Staubli VAL3: FloatToBytes.pgx

program FloatToBytes(num valIn, num& hByte, num& lByte)
  local num int
begin
//*******************************************************************************
//*   ______
//*  / _____) /|
//* | |      / /
//* | | /\  / /
//* | | \ \/ /  _      Copyright (c) KEOLABS, 2016
//* | |  \__/  | |        http://www.keolabs.com
//* | |________| |
//*  \__________/
//*
//********************************************************************************
//*@file          : FloatToBytes
//*@author        : Yves Ragot
//*@version       : $Id: FloatToBytes.pgx 1558 2017-01-05 08:13:36Z yves $
//*@brief         : convert 1 float to 2 bytes
//*
//*******************************************************************************/

 valIn = round(valIn)

 hByte = roundDown(valIn / 256)
 lByte = bAnd(valIn, 255)

end
